TYPE ST_Option :
STRUCT
	series: ARRAY[0..2] OF ST_series;	
END_STRUCT
END_TYPE

(* stored: Version 1.1.0.1, ProductVersion 3.1.4022.12
   DUT ST_Option: Id {63c4ffc3-f312-4143-b9b3-14f5c5fee3e2} *)
